(* IEC 61131-3 sources: Twincat/PLC/POUs/Functions, 2 files *)

(* ---- F_CalculateAverage.st ---- *)
(*
    Calculate Average Function
    Description: Calculates the average of an array of values
    Returns: Average value
*)

FUNCTION F_CalculateAverage : LREAL
VAR_INPUT
    aValues     : ARRAY[0..99] OF LREAL;    // Input array
    iCount      : INT;                       // Number of valid values (max 100)
END_VAR

VAR
    i           : INT;
    fSum        : LREAL := 0.0;
    iValidCount : INT;
END_VAR

// Validate count to prevent array overflow
IF iCount > 100 THEN
    iValidCount := 100;
ELSIF iCount < 0 THEN
    iValidCount := 0;
ELSE
    iValidCount := iCount;
END_IF

// Calculate sum
FOR i := 0 TO iValidCount - 1 DO
    fSum := fSum + aValues[i];
END_FOR

// Calculate average
IF iValidCount > 0 THEN
    F_CalculateAverage := fSum / INT_TO_LREAL(iValidCount);
ELSE
    F_CalculateAverage := 0.0;
END_IF

(* ---- F_ScaleValue.st ---- *)
(*
    Scale Value Function
    Description: Scales a value from one range to another
    Returns: Scaled value
*)

FUNCTION F_ScaleValue : LREAL
VAR_INPUT
    fInputValue     : LREAL;    // Value to scale
    fInputMin       : LREAL;    // Input minimum
    fInputMax       : LREAL;    // Input maximum
    fOutputMin      : LREAL;    // Output minimum
    fOutputMax      : LREAL;    // Output maximum
END_VAR

VAR
    fInputRange     : LREAL;
    fOutputRange    : LREAL;
    fNormalizedValue : LREAL;
END_VAR

// Calculate ranges
fInputRange := fInputMax - fInputMin;
fOutputRange := fOutputMax - fOutputMin;

// Avoid division by zero
IF ABS(fInputRange) < 0.0001 THEN
    F_ScaleValue := fOutputMin;
    RETURN;
END_IF

// Normalize input value to 0-1 range
fNormalizedValue := (fInputValue - fInputMin) / fInputRange;

// Scale to output range
F_ScaleValue := fOutputMin + (fNormalizedValue * fOutputRange);

// Clamp to output range
IF F_ScaleValue < fOutputMin THEN
    F_ScaleValue := fOutputMin;
ELSIF F_ScaleValue > fOutputMax THEN
    F_ScaleValue := fOutputMax;
END_IF
